SUBAPPLICATION TimedFunc (* Subapplication Type *)
  (* Standard: 61499-2 *)
  (* Version 1.0, 2023-01-29, Franz *)
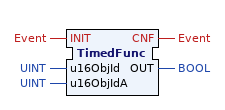
  EVENT_INPUT
    INIT;
  END_EVENT
  EVENT_OUTPUT
    CNF;
  END_EVENT
  VAR_INPUT
    u16ObjId : UINT;
    u16ObjIdA : UINT;
  END_VAR
  VAR_OUTPUT
    OUT : BOOL;
  END_VAR
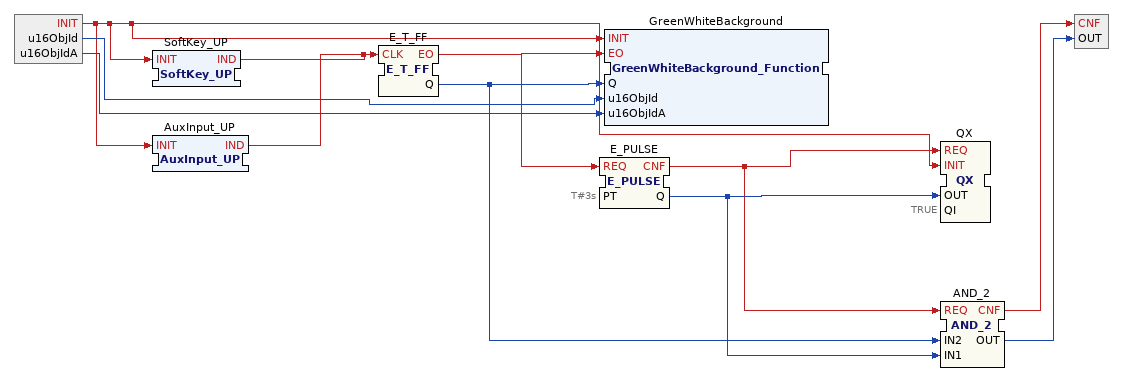
  FBS
    AND_2 : AND_2;
    E_T_FF : E_T_FF;
    QX : QX(QI := TRUE);
    E_PULSE : E_PULSE(PT := T#3s);
  END_FBS
  SUBAPPS
    GreenWhiteBackground : GreenWhiteBackground_Function;
    AuxInput_UP : AuxInput_UP;
    SoftKey_UP : SoftKey_UP;
  END_SUBAPPS
  EVENT_CONNECTIONS
    E_PULSE.CNF TO AND_2.REQ;
    E_T_FF.EO TO E_PULSE.REQ;
    E_PULSE.CNF TO QX.REQ;
    AND_2.CNF TO CNF;
    INIT TO QX.INIT;
    INIT TO GreenWhiteBackground.INIT;
    E_T_FF.EO TO GreenWhiteBackground.EO;
    INIT TO AuxInput_UP.INIT;
    AuxInput_UP.IND TO E_T_FF.CLK;
    INIT TO SoftKey_UP.INIT;
    SoftKey_UP.IND TO E_T_FF.CLK;
  END_CONNECTIONS
  DATA_CONNECTIONS
    E_T_FF.Q TO AND_2.IN2; (* Schieber offen *)
    AND_2.OUT TO OUT;
    E_T_FF.Q TO GreenWhiteBackground.Q;
    u16ObjId TO GreenWhiteBackground.u16ObjId;
    u16ObjIdA TO GreenWhiteBackground.u16ObjIdA;
    E_PULSE.Q TO QX.OUT;
    E_PULSE.Q TO AND_2.IN1;
  END_CONNECTIONS
END_SUBAPPLICATION
